KUKA KRL data list: PuxaReceita.dat

&ACCESS RV1
DEFDAT PuxaReceita

ENDDAT
